Staubli VAL3: ThrottleLogMsg.dtx

public string sMsg
public num nSeverity
public num nLastLogTime
public num nThrottleInterval
public num nMsgCountSinceLastLog
